// TIA Portal V20 export
DATA_BLOCK "DB_Maintenances"   // DB20
// stored: InstanceOfName FB_Maintenances, InstanceOfType FB
"FB_Maintenances"
   // VAR
   //    sCheckMachine : "FB_Maintenance";
   //    sReplaceAirConditioningFilter { S7_SetPoint := 'True'} : "FB_Maintenance";
   //    sMachineCooling_ReplaceWaterFilter { S7_SetPoint := 'True'} : "FB_Maintenance";
   //    sTermotekChiller_ChangeFilterAndWater { S7_SetPoint := 'True'} : "FB_Maintenance";
   //    sCheckSafetySystem { S7_SetPoint := 'True'} : "FB_Maintenance";
   //    sReplaceTipShellPeekGripper { S7_SetPoint := 'True'} : "FB_Maintenance";
   //    sReplaceFiltersVacuumLoadingUnloading { S7_SetPoint := 'True'} : "FB_Maintenance";
   //    sReplaceFiltersVacuumGenerator { S7_SetPoint := 'True'} : "FB_Maintenance";
   //    sReplaceFilterAirDryer { S7_SetPoint := 'True'} : "FB_Maintenance";
   //    sReplace5umFilter { S7_SetPoint := 'True'} : "FB_Maintenance";
   //    sReplace01umFilter { S7_SetPoint := 'True'} : "FB_Maintenance";
   //    sReplaceActiveCarbonFilter { S7_SetPoint := 'True'} : "FB_Maintenance";
   //    sUTLExtraction_ReplaceParticleFilter { S7_SetPoint := 'True'} : "FB_Maintenance";
   //    sUTLExtraction_ReplaceFilterCassetteAndActiveCarbonFilter { S7_SetPoint := 'True'} : "FB_Maintenance";
   //    sReplaceSealOnSas { S7_SetPoint := 'True'} : "FB_Maintenance";
   //    sGreaseAxes { S7_SetPoint := 'True'} : "FB_Maintenance";
   //    sMaintenance_16 { S7_SetPoint := 'True'} : "FB_Maintenance";
   //    sMaintenance_17 { S7_SetPoint := 'True'} : "FB_Maintenance";
   //    sMaintenance_18 { S7_SetPoint := 'True'} : "FB_Maintenance";
   //    sMaintenance_19 { S7_SetPoint := 'True'} : "FB_Maintenance";
   //    sMaintenance_20 { S7_SetPoint := 'True'} : "FB_Maintenance";
   //    sMaintenance_21 { S7_SetPoint := 'True'} : "FB_Maintenance";
   //    sMaintenance_22 { S7_SetPoint := 'True'} : "FB_Maintenance";
   //    sMaintenance_23 { S7_SetPoint := 'True'} : "FB_Maintenance";
   //    sMaintenance_24 { S7_SetPoint := 'True'} : "FB_Maintenance";
   //    sMaintenance_25 { S7_SetPoint := 'True'} : "FB_Maintenance";
   //    sMaintenance_26 { S7_SetPoint := 'True'} : "FB_Maintenance";
   //    sMaintenance_27 { S7_SetPoint := 'True'} : "FB_Maintenance";
   //    sMaintenance_28 { S7_SetPoint := 'True'} : "FB_Maintenance";
   //    sMaintenance_29 { S7_SetPoint := 'True'} : "FB_Maintenance";
   //    sMaintenance_30 { S7_SetPoint := 'True'} : "FB_Maintenance";
   //    sMaintenance_31 { S7_SetPoint := 'True'} : "FB_Maintenance";
   //    sMaintenance_32 { S7_SetPoint := 'True'} : "FB_Maintenance";
   //    sMaintenance_33 { S7_SetPoint := 'True'} : "FB_Maintenance";
   //    sMaintenance_34 { S7_SetPoint := 'True'} : "FB_Maintenance";
   //    sMaintenance_35 { S7_SetPoint := 'True'} : "FB_Maintenance";
   //    sMaintenance_36 { S7_SetPoint := 'True'} : "FB_Maintenance";
   //    sMaintenance_37 { S7_SetPoint := 'True'} : "FB_Maintenance";
   //    sMaintenance_38 { S7_SetPoint := 'True'} : "FB_Maintenance";
   //    sMaintenance_39 { S7_SetPoint := 'True'} : "FB_Maintenance";
   //    sMaintenance_40 { S7_SetPoint := 'True'} : "FB_Maintenance";
   //    sMaintenance_41 { S7_SetPoint := 'True'} : "FB_Maintenance";
   //    sMaintenance_42 { S7_SetPoint := 'True'} : "FB_Maintenance";
   //    sMaintenance_43 { S7_SetPoint := 'True'} : "FB_Maintenance";
   //    sMaintenance_44 { S7_SetPoint := 'True'} : "FB_Maintenance";
   //    sMaintenance_45 { S7_SetPoint := 'True'} : "FB_Maintenance";
   //    sMaintenance_46 { S7_SetPoint := 'True'} : "FB_Maintenance";
   //    sMaintenance_47 { S7_SetPoint := 'True'} : "FB_Maintenance";
   //    sMaintenance_48 { S7_SetPoint := 'True'} : "FB_Maintenance";
   //    sMaintenance_49 { S7_SetPoint := 'True'} : "FB_Maintenance";
   //    sMaintenance_50 { S7_SetPoint := 'True'} : "FB_Maintenance";
   //    sMaintenance_51 { S7_SetPoint := 'True'} : "FB_Maintenance";
   //    sMaintenance_52 { S7_SetPoint := 'True'} : "FB_Maintenance";
   //    sMaintenance_53 { S7_SetPoint := 'True'} : "FB_Maintenance";
   //    sMaintenance_54 { S7_SetPoint := 'True'} : "FB_Maintenance";
   //    sMaintenance_55 { S7_SetPoint := 'True'} : "FB_Maintenance";
   //    sMaintenance_56 { S7_SetPoint := 'True'} : "FB_Maintenance";
   //    sMaintenance_57 { S7_SetPoint := 'True'} : "FB_Maintenance";
   //    sMaintenance_58 { S7_SetPoint := 'True'} : "FB_Maintenance";
   //    sMaintenance_59 { S7_SetPoint := 'True'} : "FB_Maintenance";
   //    sMaintenance_60 { S7_SetPoint := 'True'} : "FB_Maintenance";
   //    sMaintenance_61 { S7_SetPoint := 'True'} : "FB_Maintenance";
   //    sMaintenance_62 { S7_SetPoint := 'True'} : "FB_Maintenance";
   //    sMaintenance_63 { S7_SetPoint := 'True'} : "FB_Maintenance";
   // END_VAR
BEGIN
   sCheckMachine.sElement.RunTimeSec := 0.0;
   sCheckMachine.sElement.WarningThreshold := 160;
   sCheckMachine.sElement.AlarmThreshold := 200;
   sReplaceAirConditioningFilter.sElement.RunTimeSec := 0.0;
   sReplaceAirConditioningFilter.sElement.WarningThreshold := 800;
   sReplaceAirConditioningFilter.sElement.AlarmThreshold := 1000;
   sMachineCooling_ReplaceWaterFilter.sElement.WarningThreshold := 800;
   sMachineCooling_ReplaceWaterFilter.sElement.AlarmThreshold := 1000;
   sTermotekChiller_ChangeFilterAndWater.sElement.WarningThreshold := 1600;
   sTermotekChiller_ChangeFilterAndWater.sElement.AlarmThreshold := 2000;
   sCheckSafetySystem.sElement.WarningThreshold := 1600;
   sCheckSafetySystem.sElement.AlarmThreshold := 2000;
   sReplaceTipShellPeekGripper.sElement.WarningThreshold := 1600;
   sReplaceTipShellPeekGripper.sElement.AlarmThreshold := 2000;
   sReplaceFiltersVacuumLoadingUnloading.sElement.WarningThreshold := 2400;
   sReplaceFiltersVacuumLoadingUnloading.sElement.AlarmThreshold := 3000;
   sReplaceFiltersVacuumGenerator.sElement.WarningThreshold := 2400;
   sReplaceFiltersVacuumGenerator.sElement.AlarmThreshold := 3000;
   sReplaceFilterAirDryer.sElement.WarningThreshold := 3200;
   sReplaceFilterAirDryer.sElement.AlarmThreshold := 4000;
   sReplace5umFilter.sElement.WarningThreshold := 3200;
   sReplace5umFilter.sElement.AlarmThreshold := 4000;
   sReplace01umFilter.sElement.WarningThreshold := 3200;
   sReplace01umFilter.sElement.AlarmThreshold := 4000;
   sReplaceActiveCarbonFilter.sElement.WarningThreshold := 3200;
   sReplaceActiveCarbonFilter.sElement.AlarmThreshold := 4000;
   sUTLExtraction_ReplaceParticleFilter.sElement.WarningThreshold := 3200;
   sUTLExtraction_ReplaceParticleFilter.sElement.AlarmThreshold := 4000;
   sUTLExtraction_ReplaceFilterCassetteAndActiveCarbonFilter.sElement.WarningThreshold := 3200;
   sUTLExtraction_ReplaceFilterCassetteAndActiveCarbonFilter.sElement.AlarmThreshold := 4000;
   sReplaceSealOnSas.sElement.WarningThreshold := 4800;
   sReplaceSealOnSas.sElement.AlarmThreshold := 6000;
   sGreaseAxes.sElement.WarningThreshold := 4800;
   sGreaseAxes.sElement.AlarmThreshold := 6000;
END_DATA_BLOCK
